(* CODESYS project CAN.20210529.1.project

Project tree, tasks and I/O mapping:
  Device : Changsha-Cyber-MI-linux, Changsha Cyber-MI Co., Ltd., version 3.5.10.40
    application Application
      libraries: Standard, * (System); SysFile, 3.5.15.0 (System); SysTypes2 Interfaces, * (System); SysShm, * (System); CAA Mathematics, * (CAA Technical Workgroup); SysTime, 3.5.9.0 (System); CAA Types Extern, 3.5.13.0 (CAA Technical Workgroup); CAA DTUtil Extern, 3.5.12.0 (CAA Technical Workgroup); Util, * (System); TCP, 3.5.15.0 (3S - Smart Software Solutions GmbH); CAA Net Base Services, 3.5.15.0 (CAA Technical Workgroup); MIC7001 base library, 1.1 (Cyber-MI.com); CAA SerialCom, 3.5.15.0 (CAA Technical Workgroup); CAN API, 1.0.0.3 (3S - Smart Software Solutions GmbH)
      task task_fast (cyclic, interval 20 ms, priority 10, watchdog 300 ms x 10) calls prg_can1_cfc, prg_can0_st
      programs/
        program prg_can1_cfc [CFC]: recv, send
        program prg_can0_st [ST]
    IoDrvMIC7001 : IoDrvMIC7001, Cyber-MI, version 19.1.1
        unmapped channels: Ai00@C16, Ai01@C28, Ai02@C17, Ai03@C29, Ai04@C30, Ai05@C19, Ai06@C31, Ai07@C20, Ai08@C18, Ai09@D18, Ai10@D20, Ai11@D31, Ai12@D19, Ai13@D30, Ai14@D29, Ai15@D17, Ai16@D28, Ai17@D16, Ai18-Do00@C25, Ai19-Do01@C24, Ai20-Do02@C13, Ai21-Do03@C01, Ai22-Do04@C03, Ai23-Do05@C04, Ai24-Do06@C05, Ai25-Do07@C06, Ai26-Do08@C08, Ai27-Do09@C09, Ai28-Do10@C10, Ai29-Do11@C11, Ai30-Do12@D34, Ai31-Do13@D35, Ai32-Do14@D23, Ai33-Do15@D12, Ai34-Do16@D10, Ai35-Do17@D09, Ai36-Do18@D08, Ai37-Do19@D07, Ai38-Do20@D05, Ai39-Do21@D04,
          Ai40-Do22@D03, Ai41-Do23@D02, Ai42-Do24@C23, Ai43-Do25@C35, Ai44-Do26@D24, Ai45-Do27@D13, Ai46-Ao00@C22, Ai47-Ao01@D14, Ai48_Pi02, Ai49_Out5V, Ai50_VCC, Ai51_VCC_L, Ai52_VCC_R, Ai53_Pwm-i0, Ai54_Pwm-i1, Ai55_Pwm-i2, Ai56_Pwm-i3, Ai57_CPU-T, Ai58_G-x, Ai59_G-y, Ai60_G-z, Ai61-reserved, Ai62-IO-cntr, Ai63-CDS-cntr, Di00-Ai00@C16, Di01-Ai01@C28, Di02-Ai02@C17, Di03-Ai03@C29, Di04-Ai04@C30, Di05-Ai05@C19, Di06-Ai06@C31, Di07-Ai07@C20, Di08-Ai08@C18, Di09-Ai09@D18, Di10-Ai10@D20, Di11-Ai11@D31, Di12-Ai12@D19, Di13-Ai13@D30, Di14-Ai14@D29, Di15-Ai15@D17,
          Di16-Ai16@D28, Di17-Ai17@D16, Di18-Ai18@C25, Di19-Ai19@C24, Di20-Ai20@C13, Di21-Ai21@C01, Di22-Ai22@C03, Di23-Ai23@C04, Di24-Ai24@C05, Di25-Ai25@C06, Di26-Ai26@C08, Di27-Ai27@C09, Di28-Ai28@C10, Di29-Ai29@C11, Di30-Ai30@D34, Di31-Ai31@D35, Di32-Ai32@D23, Di33-Ai33@D12, Di34-Ai34@D10, Di35-Ai35@D09, Di36-Ai36@D08, Di37-Ai37@D07, Di38-Ai38@D05, Di39-Ai39@D04, Di40-Ai40@D03, Di41-Ai41@D02, Di42-Ai42@C23, Di43-Ai43@C35, Di44-Ai44@D24, Di45-Ai45@D13, Di46-Ai46@C22, Di47-Ai47@D14, Di48-Pi00@C15, Di49-Pi01@C14, Di50-Pi02@D22, Di51-Pi03@D21, Di52-reserved, Di53-reserved, Di54-reserved, Di55-reserved,
          Di56-reserved, Di57-reserved, Di58-reserved, Di59-reserved, Di60-reserved, Di61-reserved, Di62-reserved, Di63-reserved, Pi00-Di48@C15, Pi01-Di49@C14, Pi02-Di50@D22, Pi03-Di51@D21, Do00-Ai18@C25, Do01-Ai19@C24, Do02-Ai20@C13, Do03-Ai21@C01, Do04-Ai22@C03, Do05-Ai23@C04, Do06-Ai24@C05, Do07-Ai25@C06, Do08-Ai26@C08, Do09-Ai27@C09, Do10-Ai28@C10, Do11-Ai29@C11, Do12-Ai30@D34, Do13-Ai31@D35, Do14-Ai32@D23, Do15-Ai33@D12, Do16-Ai34@D10, Do17-Ai35@D09, Do18-Ai36@D08, Do19-Ai37@D07, Do20-Ai38@D05, Do21-Ai39@D04, Do22-Ai40@D03, Do23-Ai41@D02, Do24-Ai42@C23, Do25-Ai43@C35, Do26-Ai44@D24, Do27-Ai45@D13,
          Do28-Pwmi00@C33, Do29-Pwmi01@C34, Do30-Pwmi02@D25, Do31-Pwmi03@D26, PWM00@C25, PWM01@C24, PWM02@C13, PWM03@C01, PWM04@C03, PWM05@C04, PWM06@C05, PWM07@C06, PWM08@C08, PWM09@C09, PWM10@C10, PWM11@C11, PWM12@D34, PWM13@D35, PWM14@D23, PWM15@D12, PWM16@D10, PWM17@D09, PWM18@D08, PWM19@D07, PWM20@D05, PWM21@D04, PWM22@D03, PWM23@D02, PWM24@C23, PWM25@C35, PWM26@D24, PWM27@D13, PWM28-Pwmi00@C33, PWM29-Pwmi01@C34, PWM30-Pwmi02@D25, PWM31-Pwmi03@D26, PWM_I_0@C33, PWM_I_1@C34, PWM_I_2@D25, PWM_I_3@D26,
          Ao00-Ai46@C22, Ao01-Ai47@D14, LED_run, LED_err, LED_usr, ctrl_ai_raw, ctrl_adjust, ctrl_adj0, ctrl_adj1, ctrl_adj2, ctrl_adj3, disable_5V
    SoftMotion General Axis Pool
  libraries: VisuSymbols, 3.5.10.0 (System)
  5ce3da45-db07-42e7-a21c-a00fff4ed8f6|C:\Users\zhou\p01.bmp
  5ce3da45-db07-42e7-a21c-a00fff4ed8f6|C:\working\p01.bmp
  5ce3da45-db07-42e7-a21c-a00fff4ed8f6|C:\working\file.bmp
  text list GlobalTextList
*)

// Device/Application/programs/prg_can1_cfc
PROGRAM prg_can1_cfc  // CAN 功能块 CFC语言例程， 需要安装 mic7001_baselib V0.96或以上版本
VAR

    reg_11bit:ARRAY[0..63] OF UDINT :=     [64(0)];  // 注册基本帧id，最多支持64个，如果不够，请联系厂家定制
    timeout_11bit:ARRAY[0..63] OF UDINT := [64(0)]; // 设置四个基本帧的接收超时时间，单位： 毫秒
    
    reg_29bit:ARRAY[0..63] OF UDINT :=     [16#181, 16#281, 62(0)];  // 注册两个扩展帧id，最多支持64个，如果不够，请联系厂家定制
    timeout_29bit:ARRAY[0..63] OF UDINT := [500,    500,    62(0)]; // 设置两个扩展帧的接收超时时间，单位： 毫秒
    
    msgSend11bit:CAN.MESSAGE;
    msgSend29bit:CAN.MESSAGE;
    
    send_123:BOOL := FALSE;  // 需要发送数据 123帧
	send_456:BOOL := FALSE;  // 需要发送数据 456帧
	
    recv_id:UDINT;
    recv_data:ARRAY[0..7] OF BYTE;
    bData:BYTE;
	
	rmt_start:BOOL; // 遥控器启动
	rmt_horn:BOOL;  // 遥控器喇叭
	
	ton_send123:ton :=(pt := T#100MS, et := T#5MS);  // 发送定时器
	ton_send456:ton :=(pt := T#100MS, et := T#75MS);  // 发送定时器
	FB_CAN1_A1A4_0:MIC7001_BASE.FB_CAN1_A1A4;
END_VAR

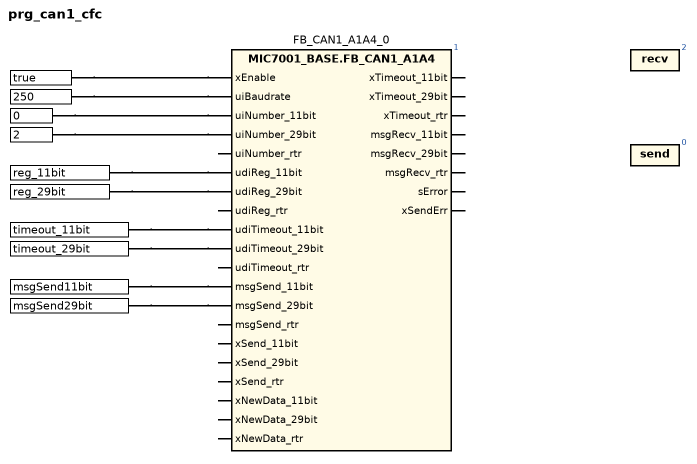
send();
FB_CAN1_A1A4_0(
    xEnable := true,
    uiBaudrate := 250,
    uiNumber_11bit := 0,
    uiNumber_29bit := 2,
    udiReg_11bit := reg_11bit,
    udiReg_29bit := reg_29bit,
    udiTimeout_11bit := timeout_11bit,
    udiTimeout_29bit := timeout_29bit,
    msgSend_11bit := msgSend11bit,
    msgSend_29bit := msgSend29bit); // MIC7001_BASE.FB_CAN1_A1A4
recv();

ACTION recv:

IF FB_CAN1_A1A4_0.xNewData_29bit[0] THEN   // 收到 181
    // 接收数据
    recv_id := FB_CAN1_A1A4_0.msgRecv_29bit[0].udiCanID;
	IF recv_id = 16#181 THEN
		//读取181帧第一个字节
		bData := FB_CAN1_A1A4_0.msgRecv_29bit[0].abyData[0];
		rmt_start := bData.0;
		rmt_horn := bData.1;
		// ... 读取其他数据
		
		// 读取181帧第二个字节
		bData := FB_CAN1_A1A4_0.msgRecv_29bit[0].abyData[1];
		// 摆臂油缸+
		// 摆臂油缸-
		// ...
		
	END_IF
	
    FB_CAN1_A1A4_0.xNewData_29bit[0] := FALSE;  // 清除新数据标志
	
ELSIF FB_CAN1_A1A4_0.xTimeout_29bit[0] THEN  // 301帧接收超时
    // 超时处理	
	
END_IF

IF FB_CAN1_A1A4_0.xNewData_29bit[1] THEN   // 收到 281
    // 接收数据
    recv_id := FB_CAN1_A1A4_0.msgRecv_29bit[1].udiCanID;
	IF recv_id = 16#281 THEN
		//读取281帧第一个字节
		bData := FB_CAN1_A1A4_0.msgRecv_29bit[0].abyData[0];
		// 转向手柄 := bData.0;
		// 伸缩手柄 := bData.1;
		// ... 读取其他数据
				
	END_IF
    
    FB_CAN1_A1A4_0.xNewData_29bit[0] := FALSE;  // 清除新数据标志
	
ELSIF FB_CAN1_A1A4_0.xTimeout_29bit[0] THEN  // 301帧接收超时
    // 超时处理	
	
END_IF
END_ACTION

ACTION send:

ton_send123(in := NOT ton_send123.Q);
IF ton_send123.Q THEN
	send_123 := TRUE;
END_IF

ton_send456(in := NOT ton_send456.Q);
IF ton_send456.Q THEN
	send_456 := TRUE;
END_IF

IF send_123 THEN
    msgSend29bit.udiCanID := 16#123;
    msgSend29bit.usiDataLength := 8;
    msgSend29bit.abyData[0] := 12; // 巡航速率对应变量
    msgSend29bit.abyData[1] := 1;  // 前方离壁距离
    msgSend29bit.abyData[2] := 23; //
    msgSend29bit.abyData[3] := 21; // 后方离壁距离
    msgSend29bit.abyData[4] := 12; // 
    msgSend29bit.abyData[5] := 45; // 夹具实时压力
    msgSend29bit.abyData[6] := 56; // 油温
    msgSend29bit.abyData[7] := 78; //
    FB_CAN1_A1A4_0.xSend_29bit := TRUE;  // 启动发送
   
    send_123 := FALSE;
END_IF

IF send_456 THEN
	msgSend29bit.udiCanID := 16#456;
    msgSend29bit.usiDataLength := 8;
    msgSend29bit.abyData[0] := 12; // 备用
    msgSend29bit.abyData[1] := 1;  // 
    msgSend29bit.abyData[2] := 0; //
    msgSend29bit.abyData[3] := 0; // 
    msgSend29bit.abyData[4] := 0; // 
    msgSend29bit.abyData[5] := 0; // 
    msgSend29bit.abyData[6] := 0; // 
    msgSend29bit.abyData[7] := 0; //	
	FB_CAN1_A1A4_0.xSend_29bit := TRUE;  // 启动发送
	send_456 := FALSE;
END_IF
END_ACTION

END_PROGRAM

// Device/Application/programs/prg_can0_st
PROGRAM prg_can0_st
VAR
	can0:MIC7001_base.FB_CAN0_B2B4;
	can11:MIC7001_base.FB_CAN1_A1A4;
	inited:BOOL := FALSE;
	msg:can.RxMESSAGE;
	rx_cntr_123:DINT := 0;
	rx_cntr_456:DINT := 0;
END_VAR


IF NOT inited THEN

	can0.m_set_baudrate(250);
	
	can0.m_reg_id_29bit(id := 16#123, timeout := 300);
	can0.m_reg_id_29bit(id := 16#456, timeout := 300);
	
	can0.m_start();
	
	inited := TRUE;
END_IF

can0();

IF can0.m_recv_msg_29bit(id := 16#123, pMsg := ADR(msg)) > 0 THEN
    rx_cntr_123 := rx_cntr_123+1;
END_IF


IF can0.m_recv_msg_29bit(id := 16#456, pMsg := ADR(msg)) > 0 THEN
 rx_cntr_456 := rx_cntr_456+1;
END_IF

END_PROGRAM
